// TIA Portal V17 export
// export: Created 2025-03-10T13:09:27.0358421Z, ExportSetting WithDefaults, DisplayName Totally Integrated Automation Portal, DisplayVersion V17 Update 8, DisplayName TIA Portal Openness, DisplayVersion V17 Update 8, DisplayName TIA Portal Version Control Interface, DisplayVersion V17, DisplayName SINAMICS Startdrive Advanced, DisplayVersion V17 SP2, DisplayName SINAMICS Startdrive G110M, G120, G120C, G120D, G120P, G115D, DisplayVersion V17 SP2, DisplayName SINAMICS Startdrive G130, G150, S120, S150, SINAMICS MV, S210, DisplayVersion V17 SP2, DisplayName STEP 7 Professional, DisplayVersion V17 Update 8, DisplayName SINUMERIK ONE STEP 7 Toolbox, DisplayVersion V17 Update 12, DisplayName SINUMERIK 840D sl STEP 7 Toolbox, DisplayVersion V17 Update 12, DisplayName STEP 7 Safety, DisplayVersion V17 Update 6, DisplayName WinCC Advanced, DisplayVersion V17 Update 8
ORGANIZATION_BLOCK "OB100_RESTART"   // OB100, LAD, Startup
TITLE = "Complete Restart"
{ S7_Optimized_Access := 'FALSE' }
AUTHOR : ETXETAR
VERSION : 1.0
// stored: AutoNumber false, IsIECCheckEnabled false, SetENOAutomatically false
   VAR_TEMP
      OB100_EV_CLASS : Byte;
      OB100_STRTUP : Byte;
      OB100_PRIORITY : Byte;
      OB100_OB_NUMBR : Byte;
      OB100_RESERVED_1 : Byte;
      OB100_RESERVED_2 : Byte;
      OB100_STOP : Word;
      OB100_RESERVED_3 : Word;
      OB100_RESERVED_4 : Word;
      OB100_DATE_TIME : Date_And_Time;
      __PlcmigTempFillBits_20B0 : Array[0..7] of Bool;
   END_VAR
BEGIN

REGION Network 1: M_ONE / ESTABLISH "LOGIC 1" BIT
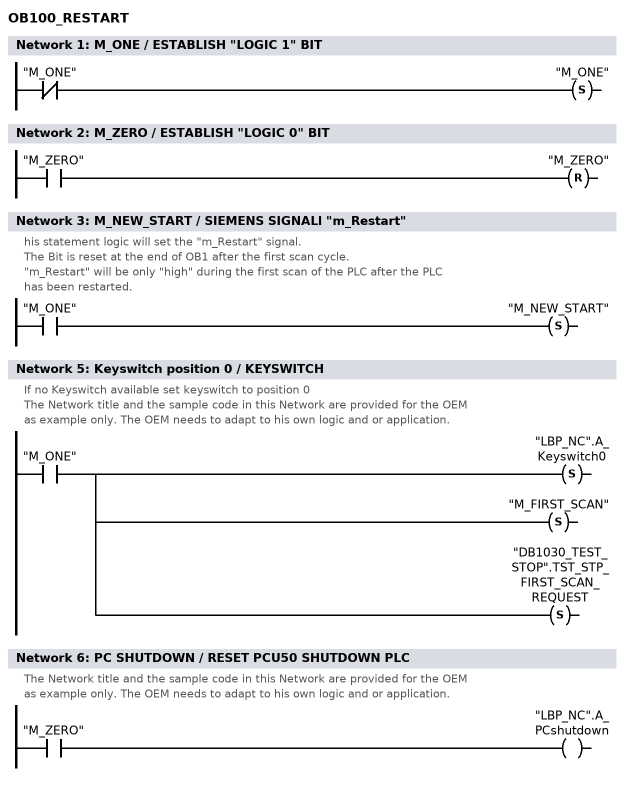
   RUNG wire#powerrail
      I_Contact( "M_ONE" )
      S_Coil( "M_ONE" )
   END_RUNG
   // the same network as SCL:
   IF NOT "M_ONE" THEN "M_ONE" := TRUE; END_IF;
END_REGION

REGION Network 2: M_ZERO / ESTABLISH "LOGIC 0" BIT
   RUNG wire#powerrail
      Contact( "M_ZERO" )
      R_Coil( "M_ZERO" )
   END_RUNG
   // the same network as SCL:
   IF "M_ZERO" THEN "M_ZERO" := FALSE; END_IF;
END_REGION

REGION Network 3: M_NEW_START / SIEMENS SIGNALl "m_Restart"
   // his statement logic will set the "m_Restart" signal.
   // The Bit is reset at the end of OB1 after the first scan cycle.
   // 
   // "m_Restart" will be only "high" during the first scan of the PLC after the PLC 
   // has been restarted.
   RUNG wire#powerrail
      Contact( "M_ONE" )
      S_Coil( "M_NEW_START" )
   END_RUNG
   // the same network as SCL:
   IF "M_ONE" THEN "M_NEW_START" := TRUE; END_IF;
END_REGION

NETWORK
TITLE = CALL FC1
      CALL  "LBP_ConfigBP"
      ( MCPNum             := 2,
        MCP1In             := "MPP_INS",
        MCP1Out            := "MPP_OUT",
        MCP1BusAdr         := 192,
        MCP1Timeout        := S5T#700MS,
        MCP2In             := "HT10_INS",
        MCP2Out            := "HT10_OUTS",
        MCP2BusAdr         := 14,
        MCP2Timeout        := S5T#700MS,
        MCP1Stop           := FALSE,
        MCP2Stop           := FALSE,
        MCP1NotSend        := FALSE,
        MCP2NotSend        := FALSE,
        MCPBusType         := B#16#55,
        HTIf               := 0,
        HTIn               := NULL,
        HTOut              := NULL,
        HTAdr              := 2,
        HTStop             := FALSE,
        HTNotSend          := FALSE,
        NCCyclTimeout      := S5T#200MS,
        NCRunupTimeout     := S5T#50S,
        ListMDecGrp        := 0,
        MMCToIF            := TRUE,
        HWheelMMC          := FALSE,
        MCP_IF_TCS         := FALSE,
        ExtendChanAxMsg    := FALSE,
        HMIAxisSel         := FALSE,
        MsgUser            := 10,
        IRAuxfuT           := FALSE,
        IRAuxfuH           := FALSE,
        IRAuxfuE           := FALSE,
        UserVersion        := "LBP_ConfigData".UserVersionInfo,
        OpKeyNum           := 0,
        Op1KeyIn           := NULL,
        Op1KeyOut          := NULL,
        Op1KeyBusAdr       := 0,
        Op2KeyIn           := NULL,
        Op2KeyOut          := NULL,
        Op2KeyBusAdr       := 0,
        Op1KeyStop         := FALSE,
        Op2KeyStop         := FALSE,
        Op1KeyNotSend      := FALSE,
        Op2KeyNotSend      := FALSE,
        OpUnitCommId       := 1,
        OpUnitInterfaceId  := 262,
        MCP1ConnectionId   := 1001,
        MCP2ConnectionId   := 1002,
        HTConnectionId     := 1003,
        Op1KeyConnectionId := 1004,
        Op2KeyConnectionId := 1005,
        IdentConnectionId  := 1006,
        MCP1LocalUdpPort   := 16001,
        MCP2LocalUdpPort   := 16002,
        HTLocalUdpPort     := 16003,
        Op1KeyLocalUdpPort := 16004,
        Op2KeyLocalUdpPort := 16005,
        IdentLocalUdpPort  := 16006,
        MaxModeGroup       := "LBP_ConfigData".MaxModeGroup,
        MaxChan            := "LBP_ConfigData".MaxChan,
        MaxAxis            := "LBP_ConfigData".MaxAxis,
        ActiveChan         := "LBP_ConfigData".ActiveChan,
        ActiveAxis         := "LBP_ConfigData".ActiveAxis,
        MaxNumUserDataInt  := "LBP_ConfigData".MaxNumUserDataInt,
        MaxNumUserDataHex  := "LBP_ConfigData".MaxNumUserDataHex,
        MaxNumUserDataReal := "LBP_ConfigData".MaxNumUserDataReal,
        UserDataIntArray   := NULL,
        UserDataHexArray   := NULL,
        UserDataRealArray  := NULL,
        TMMagazines        := NULL
      );







REGION Network 5: Keyswitch position 0 / KEYSWITCH
   // If no Keyswitch available set keyswitch to position 0
   // 
   // The Network title and the sample code in this Network are provided for the OEM 
   // as example only. The OEM needs to adapt to his own logic and or application.
   RUNG wire#powerrail
      Contact( "M_ONE" )
      wire#w1
      S_Coil( "LBP_NC".A_Keyswitch0 )
   END_RUNG
   RUNG wire#w1
      S_Coil( "M_FIRST_SCAN" )
   END_RUNG
   RUNG wire#w1
      S_Coil( "DB1030_TEST_STOP".TST_STP_FIRST_SCAN_REQUEST )
   END_RUNG
   // the same network as SCL:
   IF "M_ONE" THEN
       "LBP_NC".A_Keyswitch0 := TRUE;
       "M_FIRST_SCAN" := TRUE;
       "DB1030_TEST_STOP".TST_STP_FIRST_SCAN_REQUEST := TRUE;
   END_IF;
END_REGION

REGION Network 6: PC SHUTDOWN / RESET PCU50 SHUTDOWN PLC
   // The Network title and the sample code in this Network are provided for the OEM 
   // as example only. The OEM needs to adapt to his own logic and or application.
   RUNG wire#powerrail
      Contact( "M_ZERO" )
      Coil( "LBP_NC".A_PCshutdown )
   END_RUNG
   // the same network as SCL:
   "LBP_NC".A_PCshutdown := "M_ZERO";
END_REGION
END_ORGANIZATION_BLOCK
